(* CODESYS project CtaVisSymbols_1.0.0.1.library
   DocFormat: reStructuredText
   DefaultNamespace: CtaVisSymbols
   Version: 1.0.0.1
   Placeholder: CtaVisSymbols
   Company: CTA
   Description: Symbol Library der CTA
   CompiledLibraryCompatibilityVersion: CODESYS V3.5 SP16 Patch 3
   LanguageModelAttribute: qualified-access-only
   Title: CtaVisSymbols
   Author: SIS

Project tree, tasks and I/O mapping:
  libraries: CmpBitmapPool, 3.5.17.0 (System); VisuSymbols, 4.5.0.0 (System)
  40 Visualizations/
  30 Program Organization Units/
  00000000-0000-0000-0000-000000000000|D:\CoDeSys\LibrariesV3\trunk\Intern\CAA\CAA Template\3.4.0.0 draft\Placeholder.xml
  00000000-0000-0000-0000-000000000000|D:\CoDeSys\LibrariesV3\trunk\Intern\CAA\CAA Template\3.2.0.3 draft\Prefix.pdf
  00000000-0000-0000-0000-000000000000|D:\CoDeSys\LibrariesV3\trunk\Intern\CAA\CAA Template\3.5.2.0 draft\Placeholder.xml
  20 Structs/
  50 Images/
    image pool ImagePool
  10 Documenation/
    global variables VersionHistory
    global variables readMe
  21 Interface/
  11 Library Parameter/
  12 Konstanten/
  60 Textlisten/
  13 Globale Variablen/
  5ce3da45-db07-42e7-a21c-a00fff4ed8f6|Icons\Account.svg
  5ce3da45-db07-42e7-a21c-a00fff4ed8f6|Icons\alert.svg
  5ce3da45-db07-42e7-a21c-a00fff4ed8f6|Icons\alert_solo_black.svg
  5ce3da45-db07-42e7-a21c-a00fff4ed8f6|Icons\arrow-down.svg
  5ce3da45-db07-42e7-a21c-a00fff4ed8f6|Icons\arrow-down_solo_black.svg
  5ce3da45-db07-42e7-a21c-a00fff4ed8f6|Icons\arrow-down_square.svg
  5ce3da45-db07-42e7-a21c-a00fff4ed8f6|Icons\arrow-left.svg
  5ce3da45-db07-42e7-a21c-a00fff4ed8f6|Icons\arrow-left_solo_black.svg
  5ce3da45-db07-42e7-a21c-a00fff4ed8f6|Icons\arrow-left_square.svg
  5ce3da45-db07-42e7-a21c-a00fff4ed8f6|Icons\arrow-right_solo_black.svg
  5ce3da45-db07-42e7-a21c-a00fff4ed8f6|Icons\arrow-right_square.svg
  5ce3da45-db07-42e7-a21c-a00fff4ed8f6|Icons\arrow-up.svg
  5ce3da45-db07-42e7-a21c-a00fff4ed8f6|Icons\build.svg
  5ce3da45-db07-42e7-a21c-a00fff4ed8f6|Icons\calendar-range.svg
  5ce3da45-db07-42e7-a21c-a00fff4ed8f6|Icons\chart-bell-curve.svg
  5ce3da45-db07-42e7-a21c-a00fff4ed8f6|Icons\check.svg
  5ce3da45-db07-42e7-a21c-a00fff4ed8f6|Icons\check_solo_black.svg
  5ce3da45-db07-42e7-a21c-a00fff4ed8f6|Icons\clock-outline.svg
  5ce3da45-db07-42e7-a21c-a00fff4ed8f6|Icons\close.svg
  5ce3da45-db07-42e7-a21c-a00fff4ed8f6|Icons\close_solo_black.svg
  5ce3da45-db07-42e7-a21c-a00fff4ed8f6|Icons\CtaError.svg
  5ce3da45-db07-42e7-a21c-a00fff4ed8f6|Icons\CtaInfo.svg
  5ce3da45-db07-42e7-a21c-a00fff4ed8f6|Icons\CtaWarning.svg
  5ce3da45-db07-42e7-a21c-a00fff4ed8f6|Icons\database_black.svg
  5ce3da45-db07-42e7-a21c-a00fff4ed8f6|Icons\delete.svg
  5ce3da45-db07-42e7-a21c-a00fff4ed8f6|Icons\delete_solo_black.svg
  5ce3da45-db07-42e7-a21c-a00fff4ed8f6|Icons\dip-switch.svg
  5ce3da45-db07-42e7-a21c-a00fff4ed8f6|Icons\engine.svg
  5ce3da45-db07-42e7-a21c-a00fff4ed8f6|Icons\eye.svg
  5ce3da45-db07-42e7-a21c-a00fff4ed8f6|Icons\front_hand_Black.svg
  5ce3da45-db07-42e7-a21c-a00fff4ed8f6|Icons\front_hand_Yellow.svg
  5ce3da45-db07-42e7-a21c-a00fff4ed8f6|Icons\front_hand_Yellow_Off.svg
  5ce3da45-db07-42e7-a21c-a00fff4ed8f6|Icons\functions_black_24dp.svg
  5ce3da45-db07-42e7-a21c-a00fff4ed8f6|Icons\gear.svg
  5ce3da45-db07-42e7-a21c-a00fff4ed8f6|Icons\help.svg
  5ce3da45-db07-42e7-a21c-a00fff4ed8f6|Icons\home.svg
  5ce3da45-db07-42e7-a21c-a00fff4ed8f6|Icons\home_solo_black.svg
  5ce3da45-db07-42e7-a21c-a00fff4ed8f6|Icons\information-variant.svg
  5ce3da45-db07-42e7-a21c-a00fff4ed8f6|Icons\lan.svg
  5ce3da45-db07-42e7-a21c-a00fff4ed8f6|Icons\lightning-bolt-circle.svg
  5ce3da45-db07-42e7-a21c-a00fff4ed8f6|Icons\menu.svg
  5ce3da45-db07-42e7-a21c-a00fff4ed8f6|Icons\message.svg
  5ce3da45-db07-42e7-a21c-a00fff4ed8f6|Icons\message-alert-variant red.svg
  5ce3da45-db07-42e7-a21c-a00fff4ed8f6|Icons\message-alert-variant.svg
  5ce3da45-db07-42e7-a21c-a00fff4ed8f6|Icons\minus.svg
  5ce3da45-db07-42e7-a21c-a00fff4ed8f6|Icons\minus_solo_black.svg
  5ce3da45-db07-42e7-a21c-a00fff4ed8f6|Icons\plus.svg
  5ce3da45-db07-42e7-a21c-a00fff4ed8f6|Icons\plus_solo_black.svg
  5ce3da45-db07-42e7-a21c-a00fff4ed8f6|Icons\power.svg
  5ce3da45-db07-42e7-a21c-a00fff4ed8f6|Icons\power_solo_black.svg
  5ce3da45-db07-42e7-a21c-a00fff4ed8f6|Icons\refresh.svg
  5ce3da45-db07-42e7-a21c-a00fff4ed8f6|Icons\refresh_solo_black.svg
  5ce3da45-db07-42e7-a21c-a00fff4ed8f6|Icons\sd_card_black_24dp.svg
  5ce3da45-db07-42e7-a21c-a00fff4ed8f6|Icons\SearchFilter.svg
  5ce3da45-db07-42e7-a21c-a00fff4ed8f6|Icons\settings.svg
  5ce3da45-db07-42e7-a21c-a00fff4ed8f6|Icons\signal-celular-alt.svg
  5ce3da45-db07-42e7-a21c-a00fff4ed8f6|Icons\sine-wave.svg
  5ce3da45-db07-42e7-a21c-a00fff4ed8f6|Icons\toggle-switch.svg
  5ce3da45-db07-42e7-a21c-a00fff4ed8f6|Icons\toggle-switch-off.svg
  5ce3da45-db07-42e7-a21c-a00fff4ed8f6|Icons\Modbus_Organization_Logo.svg
  5ce3da45-db07-42e7-a21c-a00fff4ed8f6|Icons\CheckboxChecked_blue.svg
  5ce3da45-db07-42e7-a21c-a00fff4ed8f6|Icons\CheckboxUnchecked_withe.svg
  5ce3da45-db07-42e7-a21c-a00fff4ed8f6|Icons\lock_closed_black.svg
  5ce3da45-db07-42e7-a21c-a00fff4ed8f6|Icons\lock_open_black.svg
  5ce3da45-db07-42e7-a21c-a00fff4ed8f6|Icons\check_green.svg
  5ce3da45-db07-42e7-a21c-a00fff4ed8f6|Icons\close_red.svg
  5ce3da45-db07-42e7-a21c-a00fff4ed8f6|Icons\Sensor_Black.svg
  5ce3da45-db07-42e7-a21c-a00fff4ed8f6|Icons\filter_black.svg
  5ce3da45-db07-42e7-a21c-a00fff4ed8f6|Icons\notification_black.svg
  5ce3da45-db07-42e7-a21c-a00fff4ed8f6|Icons\CtaLogo.png
  5ce3da45-db07-42e7-a21c-a00fff4ed8f6|Icons\Edit_Stift.svg
  5ce3da45-db07-42e7-a21c-a00fff4ed8f6|Icons\Grafana_Logo.svg
  5ce3da45-db07-42e7-a21c-a00fff4ed8f6|Icons\InfluxDb_Logo.svg
  5ce3da45-db07-42e7-a21c-a00fff4ed8f6|Icons\hourglass_top.svg
  5ce3da45-db07-42e7-a21c-a00fff4ed8f6|Icons\Settings+.svg
  5ce3da45-db07-42e7-a21c-a00fff4ed8f6|Icons\Hourglass.gif
  5ce3da45-db07-42e7-a21c-a00fff4ed8f6|Icons\HandTapAwake.svg
  5ce3da45-db07-42e7-a21c-a00fff4ed8f6|Icons\gear_white.svg
  5ce3da45-db07-42e7-a21c-a00fff4ed8f6|S:\_Temporär_SIS\CtaCodesysLibrary\01_Library\CtaVisSymbols\Icons\SettingsSmall.svg
  5ce3da45-db07-42e7-a21c-a00fff4ed8f6|S:\_Temporär_SIS\CtaCodesysLibrary\01_Library\CtaVisSymbols\Icons\FileDescription.svg
  5ce3da45-db07-42e7-a21c-a00fff4ed8f6|S:\_Temporär_SIS\CtaCodesysLibrary\01_Library\CtaVisSymbols\Icons\Modbus_Organization_Logo_Short.svg
  5ce3da45-db07-42e7-a21c-a00fff4ed8f6|S:\_Temporär_SIS\CtaCodesysLibrary\01_Library\CtaVisSymbols\Icons\Chart.svg
  5ce3da45-db07-42e7-a21c-a00fff4ed8f6|\\cta.local\mue\Daten\200_Klima_Kälte\200_300_KK_CTA_Exklusiv_Elektro\01_Elektro\03_Software\00_CtaCodesysLibrary\01_Library\CtaVisSymbols\Icons\snowflake_melting_icon.svg
*)

// 10 Documenation/VersionHistory
(* 

.. image:: ../../Images/CTA_Logo.jpg
   :align: right
   :width: 15% 

**Vorlage**   


============ =========== =========== ============================================
**Date**     **Version** **Author**  **Change**
------------ ----------- ----------- --------------------------------------------
04.03.2021   0.0.0.0     SIS         Vorlage erstellt

============ =========== =========== ============================================


*)
VAR_GLOBAL
    stInfo : STRING:= '0.0.0.0, Vorlage, CTA';
END_VAR

// 10 Documenation/readMe
(*

**ReadMe**
 
|	**Empfehlung**
|
|	Dokumentrieren Sie die Library für eine nachhaltige Entwicklung
|     
| *Beispiel*
| 
| Dies ist die Vorlage Library der CTA. Erstellen Sie ihre Library anhand dieser Vorlage.
*)

VAR_GLOBAL
    xReadMeDone              :   BOOL;
END_VAR
